(* PLC project LabelFixture, CODESYS CODESYS V3.5 SP11 *)
(* stored: creationDateTime 2026-09-10T00:00:00 *)

PROGRAM LABELS
  VAR
    xGo : BOOL;
    xA : BOOL;
    oA : BOOL;
    xB : BOOL;
    xC : BOOL;
    oC : BOOL;
  END_VAR

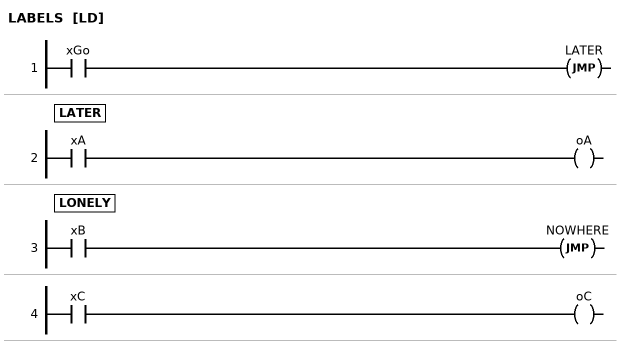
(* LD diagram, written out as Structured Text *)

IF xGo THEN JMP LATER; END_IF;

LATER:
oA := xA;

LONELY:

IF xB THEN JMP NOWHERE; END_IF;

oC := xC;
END_PROGRAM
